{attribute 'GeneratedUsingTerminal: EL3024-0000-0019'}
{attribute addProperty BoxType "EL3024-0000-0019"}
{attribute addProperty Id "AI_Compact_Channel_1AT %I*AI_Compact_Channel_80E77D6A2AI_Compact_Channel_2AT %I*AI_Compact_Channel_80E77D6A2AI_Compact_Channel_3AT %I*AI_Compact_Channel_80E77D6A2AI_Compact_Channel_4AT %I*AI_Compact_Channel_80E77D6A2WcStateAT %I*WcState_9091E0EB2InfoDataAT %I*InfoData_32EB74EA10"}
{attribute addProperty CRC "2264099861"}
{attribute addProperty Size "20"}
TYPE EL3024_86F36C15 EXTENDS EtcSlaveTerminalBase_947E5A46 :
STRUCT
	{attribute addProperty Name "AI_Compact_Channel_1"}
	AI_Compact_Channel_1 : AI_Compact_Channel_80E77D6A;
	{attribute addProperty Name "AI_Compact_Channel_2"}
	AI_Compact_Channel_2 : AI_Compact_Channel_80E77D6A;
	{attribute addProperty Name "AI_Compact_Channel_3"}
	AI_Compact_Channel_3 : AI_Compact_Channel_80E77D6A;
	{attribute addProperty Name "AI_Compact_Channel_4"}
	AI_Compact_Channel_4 : AI_Compact_Channel_80E77D6A;
	{attribute addProperty Name "WcState"}
	WcState : WcState_9091E0EB;
	{attribute addProperty Name "InfoData"}
	InfoData : InfoData_32EB74EA;
END_STRUCT
END_TYPE

(* stored: Version 1.2.0.0, ProductVersion 3.1.4024.9
   DUT EL3024_86F36C15: Id {38615859-b6eb-4a3e-beea-0e8e4ed13954} *)
